// TwinCAT 3 PLC project Untitled1_1
// ProgramVersion: 3.1.4023.0
// libraries:
//   Tc2_Standard, * (Beckhoff Automation GmbH)
//   Tc2_System, * (Beckhoff Automation GmbH)
//   Tc3_Module, * (Beckhoff Automation GmbH)
// project tree:
//   Abstract Factory/ FB_AbstractFactory.TcPOU (not stored)
//   / ClassDiagram_1.TcCD (not stored), PlcTask.TcTTO (not stored)
//   Colors/ FB_Black.TcPOU (not stored), FB_Red.TcPOU (not stored), FB_Yellow.TcPOU (not stored)
//   Creator/ FB_ShapeCreator.TcPOU, FB_ShapeCreatorEX.TcPOU, FB_ColorCreator.TcPOU (not stored)
//   DUTs/ E_Color.TcDUT (not stored), E_Factory.TcDUT (not stored), E_Shape.TcDUT
//   Factory Producer/ FB_FactoryProducer.TcPOU (not stored)
//   Interfaces/ I_Color.TcIO (not stored), I_Shape.TcIO
//   POUs/ MAIN.TcPOU (not stored)
//   Shapes/ FB_Circle.TcPOU, FB_CustomShape.TcPOU, FB_Rectangle.TcPOU, FB_Square.TcPOU, FB_Star.TcPOU, FB_Triangle.TcPOU
// real-time tasks:
//   TASK PlcTask: cycle T#10ms, priority 20, ADS port 350

// ---- DUTs/E_Shape.TcDUT
{attribute 'qualified_only'}
{attribute 'strict'}
TYPE E_Shape :
(
	init := 0,
	Circle,
	Rectangle,
	Sqaure,
	Star,
	Triangle,
	end,
	Custom
);
END_TYPE

// ---- Interfaces/I_Shape.TcIO
INTERFACE I_Shape

METHOD M_Draw : BOOL
VAR_INPUT
END_VAR
END_METHOD

END_INTERFACE

// ---- Creator/FB_ShapeCreator.TcPOU
{attribute 'hide_all_locals'}
{attribute 'enable_dynamic_creation'}
FUNCTION_BLOCK FB_ShapeCreator  EXTENDS FB_AbstractFactory
VAR_INPUT
END_VAR
VAR_OUTPUT
END_VAR
VAR
      pCircle    : POINTER TO FB_Circle;
      pRectangle : POINTER TO FB_Rectangle;
      pSquare    : POINTER TO FB_Square;
      pStar      : POINTER TO FB_Star;
      pTriangle  : POINTER TO FB_Triangle;
      iShape 	 : I_Shape;
END_VAR

METHOD FB_exit : BOOL
VAR_INPUT
	bInCopyCode : BOOL; // if TRUE, the exit method is called for exiting an instance that is copied afterwards (online change).
END_VAR
IF (pCircle <> 0) THEN
  __DELETE(pCircle);
  pCircle := 0;
END_IF

IF (pRectangle <> 0) THEN
  __DELETE(pRectangle);
  pRectangle := 0;
END_IF

IF (pSquare <> 0) THEN
  __DELETE(pSquare);
  pSquare := 0;
END_IF

IF (pStar <> 0) THEN
  __DELETE(pStar);
  pStar := 0;
END_IF

IF (pTriangle <> 0) THEN
  __DELETE(pTriangle);
  pTriangle := 0;
END_IF
END_METHOD

METHOD M_GetShapeObject : I_shape
VAR_INPUT
	eShape : E_Shape;
END_VAR
CASE eShape OF
	E_Shape.Circle:
		
		//Dynamic instantiation  
		pCircle := __NEW(FB_Circle);
		iShape := pCircle^;
		
		//Return the object
		IF iShape <> 0 THEN
			M_GetShapeObject := iShape;
		END_IF
		
		//Release the memory
		IF (pCircle <> 0) THEN
			__DELETE(pCircle);
			pCircle := 0;
		END_IF
		
		eShape := E_Shape.init;
	
	E_Shape.Rectangle:
		pRectangle := __NEW(FB_Rectangle);
		iShape := pRectangle^;
		
		//Return the object
		IF iShape <> 0 THEN
			M_GetShapeObject := iShape;
		END_IF
		
		IF (pRectangle <> 0) THEN
			__DELETE(pRectangle);
			pRectangle := 0;
		END_IF
		
		eShape := E_Shape.init;	
		
	E_Shape.Sqaure:
		pSquare := __NEW(FB_Square);
		iShape := pSquare^;
		
		//Return the object
		IF iShape <> 0 THEN
			M_GetShapeObject := iShape;
		END_IF
		
		IF (pSquare <> 0) THEN
			__DELETE(pSquare);
			pSquare := 0;
		END_IF
		
		eShape := E_Shape.init;	

	E_Shape.Star:
		pStar := __NEW(FB_Star);
		iShape := pStar^;
		
		//Return the object
		IF iShape <> 0 THEN
			M_GetShapeObject := iShape;
		END_IF
		
		IF (pStar <> 0) THEN
			__DELETE(pStar);
			pStar := 0;
		END_IF
		
		eShape := E_Shape.init;	
	
	E_Shape.Triangle:
		pTriangle := __NEW(FB_Triangle);
		iShape := pTriangle^;
		
		//Return the object
		IF iShape <> 0 THEN
			M_GetShapeObject := iShape;
		END_IF
		
		IF (pTriangle <> 0) THEN
			__DELETE(pTriangle);
			pTriangle := 0;
		END_IF
		
		eShape := E_Shape.init;	
END_CASE
END_METHOD

METHOD M_ReleaseMemory : BOOL
VAR_INPUT
END_VAR
IF (pCircle <> 0) THEN
  __DELETE(pCircle);
  pCircle := 0;
END_IF

IF (pRectangle <> 0) THEN
  __DELETE(pRectangle);
  pRectangle := 0;
END_IF

IF (pSquare <> 0) THEN
  __DELETE(pSquare);
  pSquare := 0;
END_IF

IF (pStar <> 0) THEN
  __DELETE(pStar);
  pStar := 0;
END_IF

IF (pTriangle <> 0) THEN
  __DELETE(pTriangle);
  pTriangle := 0;
END_IF
END_METHOD

END_FUNCTION_BLOCK

// ---- Shapes/FB_Circle.TcPOU
{attribute 'enable_dynamic_creation'}
FUNCTION_BLOCK FB_Circle IMPLEMENTS I_Shape
VAR_INPUT
END_VAR
VAR_OUTPUT
END_VAR
VAR
END_VAR

METHOD M_Draw : BOOL
ADSLOGSTR(ADSLOG_MSGTYPE_HINT, 'Draw circle', '');
M_Draw := TRUE;
END_METHOD

END_FUNCTION_BLOCK

// ---- Shapes/FB_Rectangle.TcPOU
{attribute 'enable_dynamic_creation'}
FUNCTION_BLOCK FB_Rectangle IMPLEMENTS I_Shape
VAR_INPUT
END_VAR
VAR_OUTPUT
END_VAR
VAR
END_VAR

{warning 'Agregar implementación de método'}
METHOD M_Draw : BOOL
ADSLOGSTR(ADSLOG_MSGTYPE_HINT, 'Draw rectangle', '');
M_Draw := TRUE;
END_METHOD

END_FUNCTION_BLOCK

// ---- Shapes/FB_Square.TcPOU
{attribute 'enable_dynamic_creation'}
FUNCTION_BLOCK FB_Square IMPLEMENTS I_Shape
VAR_INPUT
END_VAR
VAR_OUTPUT
END_VAR
VAR
END_VAR

{warning 'Agregar implementación de método'}
METHOD M_Draw : BOOL
ADSLOGSTR(ADSLOG_MSGTYPE_HINT, 'Square', '');
M_Draw := TRUE;
END_METHOD

END_FUNCTION_BLOCK

// ---- Shapes/FB_Star.TcPOU
{attribute 'enable_dynamic_creation'}
FUNCTION_BLOCK FB_Star IMPLEMENTS I_Shape
VAR_INPUT
END_VAR
VAR_OUTPUT
END_VAR
VAR
END_VAR

{warning 'Agregar implementación de método'}
METHOD M_Draw : BOOL
ADSLOGSTR(ADSLOG_MSGTYPE_HINT, 'Draw Star', '');
M_Draw := TRUE;
END_METHOD

END_FUNCTION_BLOCK

// ---- Shapes/FB_Triangle.TcPOU
{attribute 'enable_dynamic_creation'}
FUNCTION_BLOCK FB_Triangle IMPLEMENTS I_Shape
VAR_INPUT
END_VAR
VAR_OUTPUT
END_VAR
VAR
END_VAR

{warning 'Agregar implementación de método'}
METHOD M_Draw : BOOL
ADSLOGSTR(ADSLOG_MSGTYPE_HINT, 'Draw Triangle', '');
M_Draw := TRUE;
END_METHOD

END_FUNCTION_BLOCK

// ---- Creator/FB_ShapeCreatorEX.TcPOU
FUNCTION_BLOCK FB_ShapeCreatorEX EXTENDS FB_ShapeCreator
VAR_INPUT
END_VAR
VAR_OUTPUT
END_VAR
VAR
	pCustomShape : POINTER TO FB_CustomShape;
END_VAR

METHOD M_GetShapeObject : I_shape
VAR_INPUT
END_VAR
IF eShape = E_Shape.Custom THEN
	
	//Dynamic instantiation  
	pCustomShape := __NEW(FB_CustomShape);
	iShape := pCustomShape^;
	
	//Return the object
	IF iShape <> 0 THEN
		M_GetShapeObject := iShape;
	END_IF
	
	//Release the memory
	IF (pCustomShape <> 0) THEN
		__DELETE(pCustomShape);
		pCustomShape := 0;
	END_IF
	
	eShape := E_Shape.init;
ELSE
	M_GetShapeObject := SUPER^.M_GetShapeObject();
END_IF
END_METHOD

END_FUNCTION_BLOCK

// ---- Shapes/FB_CustomShape.TcPOU
{attribute 'enable_dynamic_creation'} 
FUNCTION_BLOCK FB_CustomShape IMPLEMENTS I_Shape
VAR_INPUT
END_VAR
VAR_OUTPUT
END_VAR
VAR
END_VAR

{warning 'Agregar implementación de método'}
METHOD M_Draw : BOOL
ADSLOGSTR(ADSLOG_MSGTYPE_HINT, 'Draw custom shape', '');
M_Draw := TRUE;
END_METHOD

END_FUNCTION_BLOCK
